// TIA Portal V19 export
FUNCTION_BLOCK "ButtonsSafe_LB101"   // FB150, LAD
TITLE = LB101 - SAFE PUSH BUTTONS (@ Decoiler out line / Aspo in carico)
// stored: MemoryReserve 100, SetENOAutomatically false
   VAR_INPUT
      Reset_OthersPBs_Activation_IN : Bool := FALSE;
   END_VAR
   VAR_OUTPUT
      Reset_OthersPBs_Activation_OUT : Bool;
   END_VAR
   VAR
      i : Int;
      iOperation : Int;
      iConcurrentOperation : Int;
      SettingWriteDone { S7_SetPoint := 'True'} : Bool;
      PbPanel { S7_SetPoint := 'True'} : "Buttons2Hands";
      PB : Struct
         ResetAlarms : Bool;
         Decoiler1InLine : Bool;
         Decoiler2InLine : Bool;
      END_STRUCT;
   END_VAR
   VAR CONSTANT
      ITEMS : Int := 2;
      DECOILER1_INLINE : Int := 1;
      DECOILER2_INLINE : Int := 2;
   END_VAR
BEGIN

REGION Network 1 (SCL): Interlocks between operations selected
   IF "Area01".AreaInterface.ManOneShot THEN
       #SettingWriteDone := FALSE;
   END_IF;

   // Interblocco tra operazioni
   // 
   IF NOT #SettingWriteDone THEN
       #SettingWriteDone := TRUE;

       FOR #iOperation := 1 TO #ITEMS DO
           FOR #iConcurrentOperation := 1 TO #ITEMS DO
               #PbPanel.Enables[#iOperation,#iConcurrentOperation] := FALSE;
           END_FOR;
       END_FOR;



   END_IF;
END_REGION

REGION Network 2 (SCL): Buttons for Op selection
   #PbPanel.Buttons[DECOILER1_INLINE] := "LB101_Decoiler1_Pb_InLine";
   #PbPanel.Buttons[DECOILER2_INLINE] := "LB101_Decoiler2_Pb_InLine";
END_REGION

REGION Network 3 (SCL): Operation enable
   #PbPanel.OpEnabled[DECOILER1_INLINE] := #PB.Decoiler1InLine AND ("DecoilersHRot".COut.DecoilerX_InLine_CheckNext OR "DecoilersHRot".COut.Decoiler1_InLine);
   #PbPanel.OpEnabled[DECOILER2_INLINE] := #PB.Decoiler2InLine AND ("DecoilersHRot".COut.DecoilerX_InLine_CheckNext OR "DecoilersHRot".COut.Decoiler2_InLine);
END_REGION

REGION Network 4 (SCL): Operation running
   #PbPanel.OpRunning[DECOILER1_INLINE] := "DecoilersHRot".Rotation.V.ValveSts.RestInProgress OR NOT "DecoilersHRot".COut.Pivot.Standstill OR NOT "DecoilersHRot".COut.Traslation.Standstill;
   #PbPanel.OpRunning[DECOILER2_INLINE] := "DecoilersHRot".Rotation.V.ValveSts.WorkInProgress OR NOT "DecoilersHRot".COut.Pivot.Standstill OR NOT "DecoilersHRot".COut.Traslation.Standstill;
END_REGION

REGION Network 5 (SCL): Operation done
   #PbPanel.OpDone[DECOILER1_INLINE] := "DecoilersHRot".COut.Decoiler1_InLine; //AND "DecoilersHRot".COut.Translation_InPosition;
   #PbPanel.OpDone[DECOILER2_INLINE] := "DecoilersHRot".COut.Decoiler2_InLine; //AND "DecoilersHRot".COut.Translation_InPosition;
END_REGION

REGION Network 6: Main
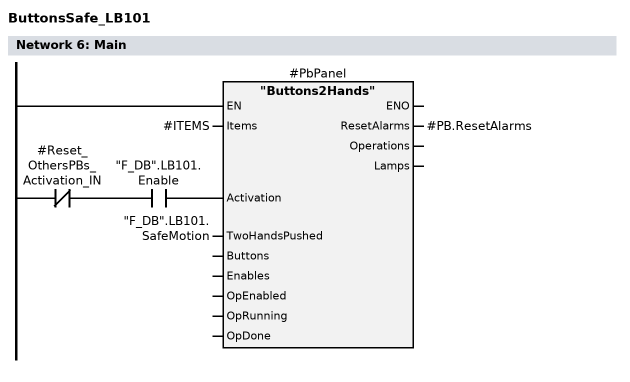
   RUNG wire#powerrail
      #PbPanel(Activation := wire#w1, Items := #ITEMS, TwoHandsPushed := "F_DB".LB101.SafeMotion, Buttons :=, Enables :=, OpEnabled :=, OpRunning :=, OpDone :=, ResetAlarms => #PB.ResetAlarms, Operations =>, Lamps =>)
   END_RUNG
   RUNG wire#powerrail
      I_Contact( #Reset_OthersPBs_Activation_IN )
      Contact( "F_DB".LB101.Enable )
   END_RUNG wire#w1
   // the same network as SCL:
   #PbPanel(Items := #ITEMS,   // "Buttons2Hands"
            Activation := NOT #Reset_OthersPBs_Activation_IN AND "F_DB".LB101.Enable,
            TwoHandsPushed := "F_DB".LB101.SafeMotion,
            ResetAlarms => #PB.ResetAlarms);
END_REGION

REGION Network 7 (SCL): Safe Buttons
   #PB.Decoiler1InLine := #PbPanel.Operations[DECOILER1_INLINE];
   #PB.Decoiler2InLine := #PbPanel.Operations[DECOILER2_INLINE];
END_REGION

REGION Network 8 (SCL): Lamp selection

   "LB101_Decoiler1_Lp_InLine" := #PbPanel.Lamps[DECOILER1_INLINE];
   "LB101_Decoiler2_Lp_InLine" := #PbPanel.Lamps[DECOILER2_INLINE];
END_REGION

REGION Network 9 (SCL): Reset others safe push buttons activation / execution
   #Reset_OthersPBs_Activation_OUT := FALSE;

   FOR #i := 1 TO #ITEMS DO

       IF #PbPanel.Buttons[#i] OR #PbPanel.Operations[#i] THEN
           #Reset_OthersPBs_Activation_OUT := TRUE;
           EXIT;
       END_IF;

   END_FOR;
END_REGION

REGION Network 10: >
END_REGION

REGION Network 11: >
END_REGION

REGION Network 12: >
END_REGION
END_FUNCTION_BLOCK
